{attribute 'no_check'}
//Returns the count of a particular char found in a string line
FUNCTION getCntCharInWStr : INT
VAR_INPUT
	Char													:	WSTRING(3):=";";
	Strline													:	WSTRING(MAX_STRING_LENGTH);
END_VAR             										
VAR                 
	tmpString												:	WSTRING(MAX_STRING_LENGTH) ;										
	pos,k													:	INT;
END_VAR

IF Strline <> "" AND Char <> ""
THEN	
	MEMSET(ADR(tmpString),0,SIZEOF(tmpString));
	MEMCPY(ADR(tmpString),ADR(Strline),TO_UDINT(WLEN(Strline) * 2));
	pos 													:= WFIND (tmpString,char);
	WHILE pos <> 0 DO		
		k													:=  pos + (WLEN(char) - 1);
		tmpString											:=	WRIGHT(tmpString,WLEN(tmpString) - k);
		pos 												:= 	WFIND (tmpString,char);
		getCntCharInWStr									:=	getCntCharInWStr+1;
	END_WHILE;
ELSE
	getCntCharInWStr										:= 0;
END_IF

END_FUNCTION

(* stored: Version 1.1.0.1, ProductVersion 3.1.4024.3
   POU getCntCharInWStr: Id {9fa268b5-472c-488f-9691-313001528ffb}, SpecialFunc None *)
